(*

short summary
=================
This is a useless interface for the validity test.

.. <legal notes>

legal notes
=================
| SPDX-FileCopyrightText: © 2024 ekvip automation GmbH <info@ekvip.de>
| SPDX-License-Identifier: Apache-2.0
| For details check: Apache-2.0_

.. _Apache-2.0: https://www.apache.org/licenses/LICENSE-2.0

.. </legal notes>

*)

INTERFACE INTERNAL IStupidObject2 EXTENDS CNM_AbstractObject.IObject

END_INTERFACE

(* stored: Version 1.1.0.1, ProductVersion 3.1.4024.12
   Itf IStupidObject2: Id {9f190e93-bbc1-4fc6-92b7-c7e86081f084} *)
